// SIMATIC S7-200 project (STEP 7-Micro/WIN), CPU 222 REL 02.01

SYMBOL_TABLE USER1
START            I0.0     // start button
STOP_            I0.1     // stop button
S1               I0.2     // Extended position of actuator 1
S2               I0.3     // Extended position of actuator 2
S3               I0.4     // Retracted psotion of Feeder actuator
S4               I0.5     // Extended position of Feeder actuator
RLBS             I0.6     // Reflex light beam sensor with reflector
ColorS           I0.7     // Color sensor to detect non-red objects
Cap              I1.0     // Capactive sensor for feeder
Conveyor         Q0.0     // Conveyor belt
Y1               Q0.1     // Extend Actuator 1
Y2               Q0.2     // Extend Actuator 2
Y3               Q0.3     // Extend Feeder
Y4               Q0.4     // Retract Feeder
END_SYMBOL_TABLE

ORGANIZATION_BLOCK MAIN:OB1
TITLE=PROGRAM COMMENTS
BEGIN
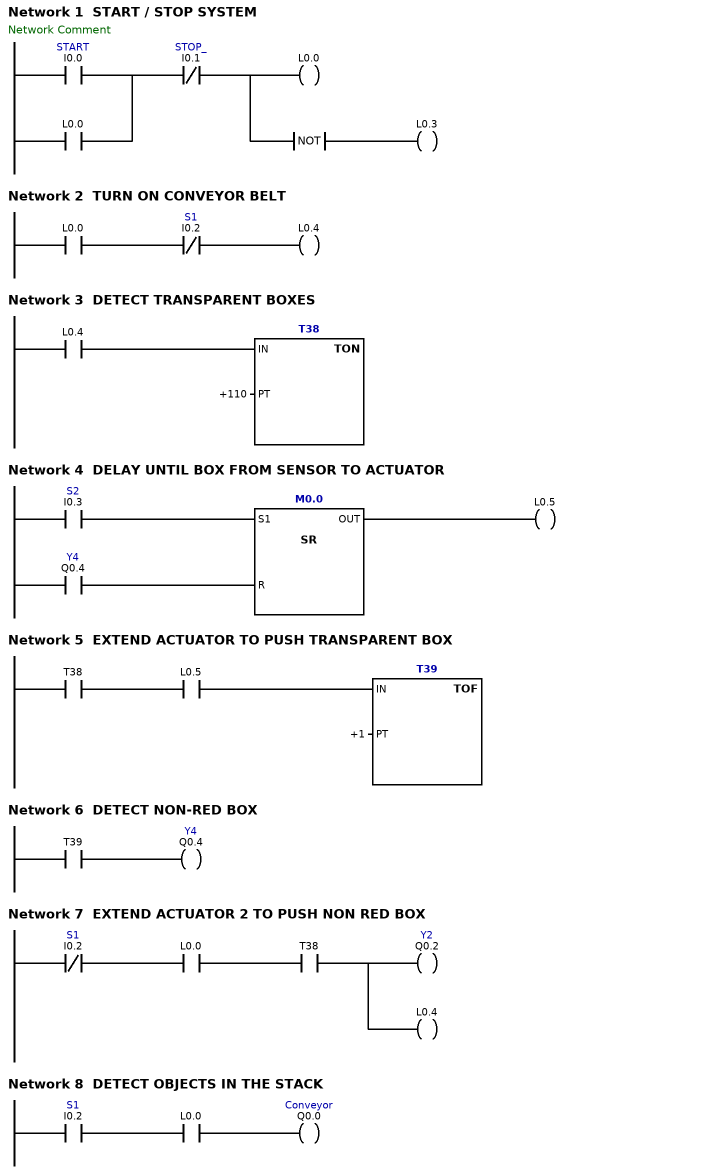
Network 1 // START / STOP SYSTEM
// Network Comment
LD     START:I0.0
O      L0.0
AN     STOP_:I0.1
=      L0.0
NOT
=      L0.3
Network 2 // TURN ON CONVEYOR BELT
LD     L0.0
AN     S1:I0.2
=      L0.4
Network 3 // DETECT TRANSPARENT BOXES 
LD     L0.4
TON    T38, +110
Network 4 // DELAY UNTIL BOX FROM SENSOR TO ACTUATOR
LD     S2:I0.3
LD     Y4:Q0.4
NOT
A      M0.0
OLD
=      M0.0
=      L0.5
Network 5 // EXTEND ACTUATOR TO PUSH TRANSPARENT BOX
LD     T38
A      L0.5
TOF    T39, +1
Network 6 // DETECT NON-RED BOX
LD     T39
=      Y4:Q0.4
Network 7 // EXTEND ACTUATOR 2 TO PUSH NON RED BOX
LDN    S1:I0.2
A      L0.0
A      T38
=      Y2:Q0.2
=      L0.4
Network 8 // DETECT OBJECTS IN THE STACK
LD     S1:I0.2
A      L0.0
=      Conveyor:Q0.0
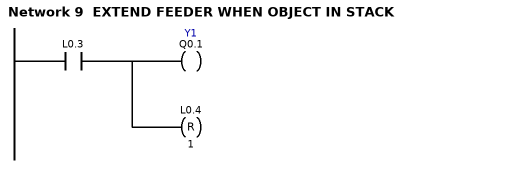
Network 9 // EXTEND FEEDER WHEN OBJECT IN STACK
LD     L0.3
=      Y1:Q0.1
R      L0.4, 1
Network 11 // RETRACT FEEDER AFTER EXTENDING
END_ORGANIZATION_BLOCK
